FUNCTION_BLOCK FB_UPS_Base
//////////////////
// UPS 
//////////////////
VAR_INPUT PERSISTENT
	// Parameters of the Object (instance/model specific) 
		ParamTimeOut					: TIME := T#2S;		(* (s) Modbus Timeout*)
		ParamClockReadTime				: TIME := T#1S;		(* (s) Modbus Reading Frequency *)
		ParamNC							: BOOL := FALSE; 	(* (NA)False: TRUE = Closed, True : TRUE = opened*)
		                                
		ParamTempoComAlarm				: TIME := T#2S;		(* (s) Tempo before raising a communication alarm*)
		ParamTempoComWarning			: TIME := T#1S;		(* (s) Tempo before raising a communication warning*)
		ParamTP_Impulsion				: TIME := T#5S;		(* (s) TP Impulsion = 5s *)
END_VAR                                 
                                        
VAR_OUTPUT                              
	//Child objects                     
		OUT_CmdRelance_IO				: BOOL;
END_VAR                                 
                                        
VAR_INPUT                               
	// I/O Inputs                       
		IN_MesDischarging_IO		  	: BOOL;
		IN_MesBatLow_IO		   			: BOOL;
		IN_MesFault_IO					: BOOL;

		IN_CmdReStartUPS				: BOOL;
		
		IN_CmdToggleRead				: BOOL;
		IN_CmdReset_L					: BOOL; 
END_VAR

VAR
	//M_ALARMMANAGEMENT VARIABLES//
		TON_ComAlarm					: TON;
		TON_ComWarning					: TON;	

		MesWarningCom					: BOOL ; 			// (NA) [P,H] True if bad modbus communication 
			
	//M_READ//
//	MesDataExd					: UPS ; 

	//M_EXECUTE //
		TP1								: TP;
		ClockRead			AT %Q*		: BOOL;
   		
    //M_CP VARIABLES//
		Trig_Cmd_Read					: R_TRIG;                                                                                        
                                                                                       
		CmdRelanceChargeur				: BOOL;
		CP_Relance						: BOOL;
		TP_Relance						: TP;
		MesCP_Read					: BOOL := TRUE;	(* Read function enable *)
		MesCP_Write					: BOOL := TRUE;	(* Write function enable *)   
END_VAR

METHOD M_AlarmManagement
//////////////////
// Manages Sepam Alarms. Alarms opens HT CB until Sepam manual Reset . Warning Opens CB-L but does not maintain warning
/////////////////

VAR 
	// Method local variables (reinitialized at each cycle) 
	FB_AlarmCodeManager 	: FB_AlarmCodeManager ; 

 
END_VAR
END_METHOD

METHOD M_Execute
//////////////////
//  Method Calls 
/////////////////

VAR 
	// Method local variables (reinitialized at each cycle) 

END_VAR


// METHODS CALLS // 
Trig_Cmd_Read(CLK:=IN_CmdToggleRead);
CP_Relance	:= IN_CmdReStartUPS ; 	
IF Trig_Cmd_Read.Q THEN
	//IN_CmdToggleRead := FALSE;
	MesCP_Read := NOT MesCP_Read;
	
END_IF

	TP1(IN:=NOT TP1.Q , PT:= ParamClockReadTime);
	ClockRead 		:= TP1.Q;

	TP_Relance(IN:= CP_Relance , PT:=ParamTP_Impulsion) ;
	OUT_CmdRelance_IO	 := TP_Relance.Q ;
	
	M_Read(); 
	M_AlarmManagement() ;
END_METHOD

METHOD M_Read
//////////////////
//  Read Modbus Variable for PCS . 
/////////////////
VAR 
	// Method local variables (reinitialized at each cycle) 
		

END_VAR
END_METHOD

END_FUNCTION_BLOCK

(* stored: Version 1.1.0.1, ProductVersion 3.1.4024.6
   POU FB_UPS_Base: Id {3666d37b-1d48-47bd-98a6-c1ac777f9c72}, SpecialFunc None
   Method M_AlarmManagement: Id {1e76f4e6-2953-429c-a3b3-a8e1579a7485}
   Method M_Execute: Id {d904a97b-4a18-4fa8-8817-af95c41483e9}
   Method M_Read: Id {bd58a7a3-3944-46e7-858a-c18b130418dd} *)
